// TwinCAT 3 PLC project my_plc_project
// ProgramVersion: 3.1.4024.0
// libraries:
//   Tc2_Standard, * (Beckhoff Automation GmbH)
//   Tc2_System, * (Beckhoff Automation GmbH)
//   Tc3_Module, * (Beckhoff Automation GmbH)
// project tree:
//   / GlobalTextList.TcGTLO, PlcTask.TcTTO, Visualization Manager.TcVMO (not stored)
//   POUs/ MAIN.TcPOU
//   VISUs/ Visualization.TcVIS
// real-time tasks:
//   TASK PlcTask: cycle T#10ms, priority 20, ADS port 350
//   TASK PlcTask1: cycle T#10ms, priority 21, ADS port 351

CONFIGURATION my_plc_project
    RESOURCE PLC ON TwinCAT3
        TASK PlcTask(INTERVAL := T#10ms, PRIORITY := 21);
        PROGRAM MAIN WITH PlcTask : MAIN;
    END_RESOURCE
END_CONFIGURATION

// ---- POUs/MAIN.TcPOU
PROGRAM MAIN
VAR
	bPizzaInOven : BOOL;
	bBuzzer : BOOL;
	fbPizzaTimer : TON;
	iTotalPizzasCooked : UDINT;
	fbMyTrigger_RTRIG : R_TRIG; // This counts the Pizza
	iHeartBeat: INT; 
END_VAR



iHeartBeat := iHeartBeat + 1;

fbPizzaTimer(IN:=bPizzaInOven,PT:=T#3S);

bBuzzer := fbPizzaTimer.Q; // bBuzzer is true when fbPizzaTimer is done.

fbMyTrigger_RTRIG(clk:=fbPizzaTimer.Q); // note to self, clk is the rising edge input param

IF fbMyTrigger_RTRIG.Q THEN
	iTotalPizzasCooked := iTotalPizzasCooked + 1;
END_IF

END_PROGRAM

// ---- GlobalTextList.TcGTLO
TEXTLIST GlobalTextList
  962 = 'Buzzer'
  50 = 'Elapsed Time: %s'
  872 = 'Insert Pizza'
  731 = 'Light'
  707 = 'Take Pizza Out'
END_TEXTLIST

// ---- VISUs/Visualization.TcVIS
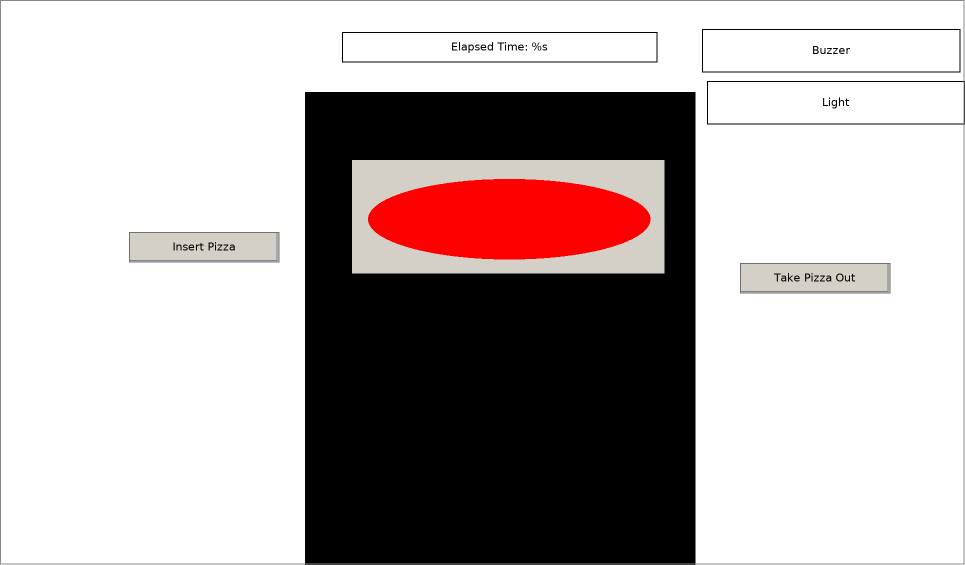
VISUALIZATION Visualization  // 965x565
    Button (129,232 150x30), "Insert Pizza"
        OnMouseClick: execute { MAIN.bPizzaInOven := TRUE; }
    Button (740,263 150x30), "Take Pizza Out"
        OnMouseClick: execute { MAIN.bPizzaInOver := False; }
    Rectangle (305,92 390x473)
    Rectangle (342,32 315x30), "Elapsed Time: %s", text variable: MAIN.fbPizzaTimer.ET
    RoundedRectangle (352,160 312x113)
    Ellipse (367,178 284x82), invisible if: NOT MAIN.bPizzaInOven
    RoundedRectangle (702,29 258x43), "Buzzer", colour toggle: MAIN.bBuzzer
    RoundedRectangle (707,81 258x43), "Light", colour toggle: MAIN.bPizzaInOven
END_VISUALIZATION
